FUNCTION_BLOCK xPPU_PAC
VAR_INPUT
	i_error: POINTER TO ErrorManager;
	i_process: POINTER TO ProcessManager;
	i_state: POINTER TO StateTracker;
END_VAR
VAR
	m_emptyParams: ParameterSet;
	m_subRes: EOperationResult;
END_VAR

VAR
	m_alarm_flags: ARRAY [1..10] OF BOOL := [FALSE, FALSE, FALSE, FALSE, FALSE, FALSE,FALSE, FALSE, FALSE, FALSE];
	m_timer_PresenceSensor: TON;
	m_errorManager: ErrorManager;
	m_services: ServiceContainer(ADR(m_errorManager));
	
	fbEndFalling   : F_TRIG;   // detect negative edge in action WPAccumulate
  	fbStartRising  : R_TRIG;   // detect positive edge in action WPAccumulate
  	tmr2s          : TON;      // 2s delay，for action WPAccumulation
  	tmr3s          : TON;      // 3s delay，for action WPAccumulation
  	po4 : BOOL;
	PAC_PoAtEnd : BOOL;
	PAC_SwitchExtended_History : BOOL := FALSE; 
	
END_VAR

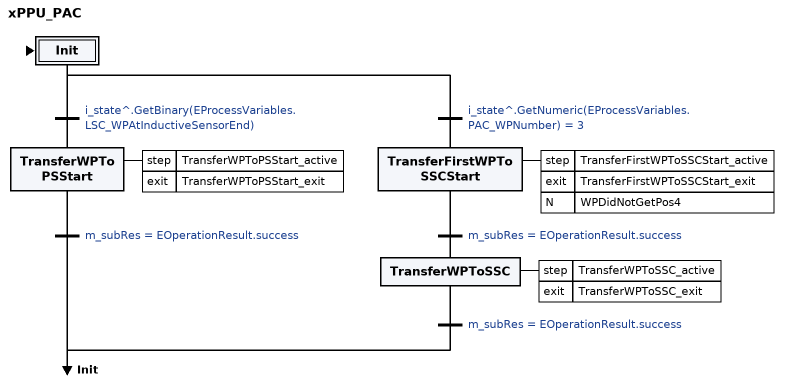
INITIAL_STEP Init:
END_STEP
TRANSITION FROM Init TO TransferWPToPSStart
    := i_state^.GetBinary(EProcessVariables.LSC_WPAtInductiveSensorEnd);
END_TRANSITION
STEP TransferWPToPSStart:
    TransferWPToPSStart_active(N);  // step action
    TransferWPToPSStart_exit(P0);  // exit action
END_STEP
TRANSITION FROM TransferWPToPSStart TO Init
    := m_subRes = EOperationResult.success;
END_TRANSITION
TRANSITION FROM Init TO TransferFirstWPToSSCStart
    := i_state^.GetNumeric(EProcessVariables.PAC_WPNumber) = 3;
END_TRANSITION
STEP TransferFirstWPToSSCStart:
    TransferFirstWPToSSCStart_active(N);  // step action
    TransferFirstWPToSSCStart_exit(P0);  // exit action
    WPDidNotGetPos4(N);
END_STEP
TRANSITION FROM TransferFirstWPToSSCStart TO TransferWPToSSC
    := m_subRes = EOperationResult.success;
END_TRANSITION
STEP TransferWPToSSC:
    TransferWPToSSC_active(N);  // step action
    TransferWPToSSC_exit(P0);  // exit action
END_STEP
TRANSITION FROM TransferWPToSSC TO Init
    := m_subRes = EOperationResult.success;
END_TRANSITION

ACTION TransferFirstWPToSSCStart_active:
m_subRes := i_process^.Execute(
	EBehaviorType.control_primitive,
	EPrimitives.PAC_TransferFitsrWorkpieceTo_SSCStart,
	m_emptyParams);
	
IF i_state^.GetBinary(EProcessVariables.PAC_SwitchExtended) THEN
    PAC_SwitchExtended_History := TRUE; 
END_IF
END_ACTION

ACTION TransferFirstWPToSSCStart_exit:
i_state^.ShiftProduct(EProducts.PAC_product1, EProducts.SSC_product1);

IF m_alarm_flags[2] = FALSE
	AND i_state^.GetNumeric(EProducts.PAC_product2) <> 0
	AND NOT i_state^.GetBinary(EProcessVariables.PAC_WPAtEnd)
THEN
    i_error^.AddMessage(EAlarms.PAC_ThirdWP_abnormal, TRUE, ESeverity.error, 'The third WP was not correctly transported on PAC');
    m_alarm_flags[2] := TRUE; 
END_IF


IF m_alarm_flags[3] = FALSE
	AND (NOT PAC_SwitchExtended_History)
	AND i_state^.GetNumeric(EProducts.PAC_product1) <> 0
	AND NOT i_state^.GetBinary(EProcessVariables.PAC_WPAtEnd)
THEN
    i_error^.AddMessage(EAlarms.PAC_FirstWP_abnormal, TRUE, ESeverity.error, 'The first WP was not correctly transported on PAC');
    m_alarm_flags[3] := TRUE;
 
END_IF

m_alarm_flags[4] := FALSE;
END_ACTION

ACTION TransferWPToPSStart_active:
m_subRes := i_process^.Execute(
	EBehaviorType.control_primitive,
	EPrimitives.PAC_TransferWorkpieceTo_PSStart,
	m_emptyParams);
END_ACTION

ACTION TransferWPToPSStart_exit:
CASE LREAL_TO_INT(i_state^.GetNumeric(EProcessVariables.PAC_WPNumber)) OF
	1:	i_state^.ShiftProduct(EProducts.LSC_product, EProducts.PAC_product1);
	2:	i_state^.ShiftProduct(EProducts.LSC_product, EProducts.PAC_product2);
	3: 	i_state^.ShiftProduct(EProducts.LSC_product, EProducts.PAC_product3);
END_CASE

IF m_alarm_flags[1] = FALSE
	AND NOT i_state^.GetBinary(EProcessVariables.PAC_WPAtStart)
THEN
    i_error^.AddMessage(EAlarms.LSC_WP_ToPAC_abnormal, TRUE, ESeverity.error, 'The first metal WP was not correctly transported to PAC Switch');
    m_alarm_flags[1] := TRUE; 
END_IF
END_ACTION

ACTION TransferWPToSSC_active:
m_subRes := i_process^.Execute(
	EBehaviorType.control_primitive,
	EPrimitives.PAC_TransferWorkpieceTo_SSC,
	m_emptyParams);
END_ACTION

ACTION TransferWPToSSC_exit:
//shift products from PAC to SSC
i_state^.ShiftProduct(EProducts.PAC_product2, EProducts.SSC_product2);
i_state^.ShiftProduct(EProducts.PAC_product3, EProducts.SSC_product3);
END_ACTION

ACTION WPDidNotGetPos4:
IF i_state^.GetBinary(EProcessVariables.PAC_SwitchExtended) 	
THEN
   	m_timer_PresenceSensor(IN := TRUE, PT := T#3000MS);
END_IF

IF i_state^.GetBinary(EProcessVariables.PAC_WPAtEnd) THEN
    m_timer_PresenceSensor(IN := FALSE,PT := T#0MS);
END_IF

IF m_alarm_flags[4] = FALSE
   	AND m_timer_PresenceSensor.Q 
THEN
    i_error^.AddMessage(EAlarms.PAC_DNGP4, TRUE, ESeverity.error, 'WP did not get positon4 in PAC');
    m_alarm_flags[4] := TRUE; 
	m_timer_PresenceSensor(IN := FALSE,PT := T#0MS);
END_IF
END_ACTION

END_FUNCTION_BLOCK

(* stored: Version 1.1.0.1
   POU xPPU_PAC: Id {31492fc4-cd6a-47c9-9b47-d0d720b462dd}, SpecialFunc None
   Action TransferFirstWPToSSCStart_active: Id {3ee7c439-6561-414f-9034-470a714accaf}
   Action TransferFirstWPToSSCStart_exit: Id {5171b752-3096-4601-a02f-5102b5cfb1fa}
   Action TransferWPToPSStart_active: Id {d68f1288-0b40-43c1-94e0-2cb29ef010b6}
   Action TransferWPToPSStart_exit: Id {e95729a1-7980-4cdb-a261-cce4fad2646c}
   Action TransferWPToSSC_active: Id {b9f26b4d-03d2-4116-99c7-0e371a34fdf6}
   Action TransferWPToSSC_exit: Id {459563bc-8582-4e63-b8e6-b2dbdd8392c2}
   Action WPDidNotGetPos4: Id {9e95ded4-404c-4170-bf90-d8060330bfbf} *)
